FUNCTION_BLOCK ABSTRACT FB_Station IMPLEMENTS IStation
VAR_INPUT
END_VAR
VAR_OUTPUT
END_VAR
VAR
	bPartPresent			AT %I* : BOOL;
	bReady					: BOOL;
	bFaulted				: BOOL;
	bBusy					: BOOL;
	
	eState					: E_StationState;
	pPartStatus				: POINTER TO ST_PartStatus;
	tmrPartPresentDelay		: TON;
END_VAR

METHOD PROTECTED ABSTRACT DoWork : BOOL
VAR_INPUT
END_VAR
END_METHOD

METHOD PUBLIC Execute : PVOID
bReady := NOT bFaulted AND NOT bBusy;

CASE eState OF
	
	E_StationState.IDLE_READY:
		
		tmrPartPresentDelay(IN:=bPartPresent, PT:=T#300MS);
		
		IF tmrPartPresentDelay.Q AND bReady THEN
			eState := E_StationState.PART_PRESENT;
		END_IF
	
	E_StationState.PART_PRESENT:
	
		bBusy := TRUE;
		eState := E_StationState.WORKING;
	
	E_StationState.WORKING:
	
		IF DoWork() THEN
			eState := E_StationState.WORK_COMPLETE;
		END_IF
		
		IF bFaulted THEN
			eState := E_StationState.FAULTED;
		END_IF
	
	E_StationState.WORK_COMPLETE:
		
		bBusy := FALSE;
		
		IF NOT bPartPresent THEN
			UpdatePartStatus();
			eState := E_StationState.IDLE_READY;
		END_IF
	
	E_StationState.FAULTED:
	
		eState := FaultHandler();

END_CASE
END_METHOD

PROPERTY Faulted : BOOL
GET
Faulted := bFaulted;
END_GET
END_PROPERTY

METHOD PROTECTED ABSTRACT FaultHandler : E_StationState
VAR_INPUT
END_VAR
END_METHOD

PROPERTY PartPresent : BOOL
GET
PartPresent := bPartPresent;
END_GET
END_PROPERTY

PROPERTY PartStatus : POINTER TO ST_PartStatus
SET
pPartStatus := PartStatus;
END_SET
END_PROPERTY

PROPERTY Ready : BOOL
GET
Ready := bReady;
END_GET
END_PROPERTY

PROPERTY State : E_StationState
GET
State := eState;
END_GET
END_PROPERTY

METHOD PROTECTED ABSTRACT UpdatePartStatus : PVOID
VAR_INPUT
END_VAR
END_METHOD

END_FUNCTION_BLOCK

(* stored: Version 1.1.0.1, ProductVersion 3.1.4024.12
   POU FB_Station: Id {bcce9771-0d87-4ec6-bb72-01c4cc53c780}, SpecialFunc None
   Method DoWork: Id {a9114007-4794-40b7-8bf1-b47079e93cdb}
   Method Execute: Id {86608ea1-fee3-4cc8-9b1f-741b9b520762}
   Property Faulted: Id {d757f652-0d46-4612-b1e6-25a1bf6add09}
   Get Get: Id {6fb07fbc-d770-4732-8083-344b75731878}
   Method FaultHandler: Id {5df141d7-690b-4cc1-93d9-a00133bb91f7}
   Property PartPresent: Id {579b6636-2123-4dee-9b87-9104c2304a5a}
   Get Get: Id {5c5be853-cbb1-4b5b-805c-b6c87325e873}
   Property PartStatus: Id {1a0e0383-f783-4cae-ba2c-db885b735f4a}
   Set Set: Id {40ccbe83-dc3f-417e-b4d1-d461a23ea222}
   Property Ready: Id {7deb4803-d4cd-42d8-bfaa-ce274def8db3}
   Get Get: Id {6cca0dd7-1af4-406d-8913-3c119b8e954b}
   Property State: Id {84ece4b5-457b-44b4-8d69-43e5b7deb721}
   Get Get: Id {e42d24d4-507b-4fb5-83ed-cad4d56d64bc}
   Method UpdatePartStatus: Id {9a6169a7-491a-413f-9af9-6e85e86923ff} *)
